FUNCTION TFPalletizerIsWorkAreaIntoZone : BOOL

VAR_INPUT
	WorkAreaZone : POINTER TO TFMachinePalletizer_WorkAreaZone;
	WorkArea : INT;
END_VAR
VAR
	n : INT;
	i : INT;
END_VAR

TFPalletizerIsWorkAreaIntoZone := FALSE;

FOR n:=1 TO MAXZONE DO
	FOR i:=1 TO MAXAREA DO
		(* Verifico se la WorkArea appartiena ad una Zona *)
		IF WorkAreaZone^.Zone[n].WorkArea[i] = WorkArea THEN
			TFPalletizerIsWorkAreaIntoZone := TRUE;
			RETURN;
		END_IF
	END_FOR
END_FOR

END_FUNCTION

(* stored: Version 1.1.0.1, ProductVersion 3.1.4024.11
   POU TFPalletizerIsWorkAreaIntoZone: Id {c19a1ee5-d5f2-48f2-a104-da79c6a4a5d9}, SpecialFunc None *)
